PROGRAM Kommunikation_Server
VAR
	Connect			:FB_ServerClientConnection;
	Connect_Local	:FB_SocketConnect;
	Send			:FB_SocketSend;
	Receive			:FB_SocketReceive;
	hServer			:T_HSERVER;
	
	sSrvNetID : T_AmsNetID := '';
	sLocalHost : STRING(15) := '147.87.210.78';
	nLocalPort : UDINT := 21;
	nMode : DWORD := LISTEN_MODE_CLOSEALL (* OR CONNECT_MODE_ENABLEDBG*);
	bEnable : BOOL := TRUE;
	
	eMode       : E_SocketAcceptMode := eACCEPT_ALL;
    sRemoteHost : T_IPv4Addr := '192.168.50.100';
    nRemotePort : UDINT := 30002;
    tReconnect  : TIME := T#5S;
	
END_VAR

VAR_INPUT
	
	
	
END_VAR

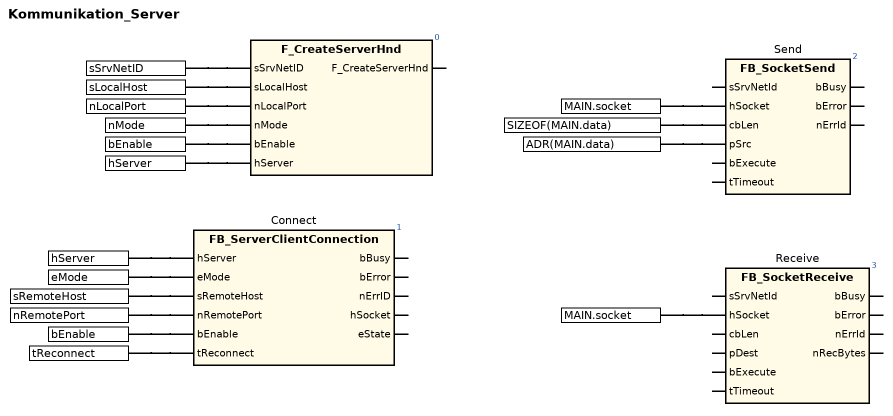
F_CreateServerHnd(sSrvNetID := sSrvNetID, sLocalHost := sLocalHost, nLocalPort := nLocalPort, nMode := nMode, bEnable := bEnable, hServer := hServer);
Connect(
    hServer := hServer,
    eMode := eMode,
    sRemoteHost := sRemoteHost,
    nRemotePort := nRemotePort,
    bEnable := bEnable,
    tReconnect := tReconnect); // FB_ServerClientConnection
Send(hSocket := MAIN.socket, cbLen := SIZEOF(MAIN.data), pSrc := ADR(MAIN.data)); // FB_SocketSend
Receive(hSocket := MAIN.socket); // FB_SocketReceive

END_PROGRAM

(* stored: Version 1.1.0.1
   POU Kommunikation_Server: Id {72a2321f-4d1d-46dc-9327-1dcc44bf5251}, SpecialFunc None *)
